TYPE ST_ELDUTTO2 :
STRUCT
	bDuttos:BOOL;
END_STRUCT
END_TYPE

(* stored: Version 1.1.0.1, ProductVersion 3.1.4024.3
   DUT ST_ELDUTTO2: Id {4e7869d3-c8e2-4864-a560-d52126ca0762} *)
